FUNCTION_BLOCK FB_Generic
VAR_INPUT
END_VAR
VAR_OUTPUT
END_VAR
VAR
END_VAR

END_FUNCTION_BLOCK

(* stored: Version 1.1.0.1, ProductVersion 3.1.4024.12
   POU FB_Generic: Id {2d1028d7-c68c-409c-9f71-89e7fa3d0153}, SpecialFunc None *)
